INTERFACE InterfaceObservable

METHOD subscribe : BOOL
VAR_INPUT
	observer : InterfaceObserver;
END_VAR
END_METHOD

END_INTERFACE

(* stored: Version 1.1.0.1, ProductVersion 3.1.4024.12
   Itf InterfaceObservable: Id {bf488430-1904-4fb9-97ea-970fa49d533c}
   Method subscribe: Id {57d1f5a3-c053-4fc8-99c4-4d8c2a1a0b81} *)
